FUNCTION_BLOCK FB_DIV_REAL (* REAL Division *)
  (* Standard: 61499-1-D.1; Classification: Math *)
  (* Version 0.0, 2001-08-05, JHC, Rockwell Automation, First implementation. *)
  (* Compiler header: package fb.rt.math; *)
  (* Compiler classdef: class FB_DIV_REAL extends FBFunctionQS2 *)
  (* Compiler Java IBM VisualAge 3.0 *)
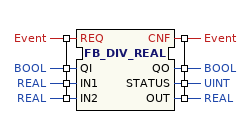
  EVENT_INPUT
    REQ WITH QI, IN1, IN2;
  END_EVENT
  EVENT_OUTPUT
    CNF WITH QO, STATUS, OUT;
  END_EVENT
  VAR_INPUT
    QI : BOOL; (* Event Qualifier *)
    IN1 : REAL; (* Dividend *)
    IN2 : REAL; (* Divisor *)
  END_VAR
  VAR_OUTPUT
    QO : BOOL; (* Output Qualifier *)
    STATUS : UINT; (* Operation Status *)
    OUT : REAL; (* Quotient *)
  END_VAR
END_FUNCTION_BLOCK
